{attribute addProperty BoxType "ELX3204-0000-0016"}
{attribute addProperty Id "RTD_Inputs_ChannelAT %I*ARRAY[0..3] OF RTD_Inputs_Channel_F16A160D128160WcStateAT %I*WcState_F855686C1620InfoDataAT %I*InfoData_BC63D37F80100"}
{attribute addProperty CRC "1009405569"}
{attribute addProperty SizeInBites "224"}
{attribute addProperty SizeInBytes "28"}
TYPE ELX3204_5DC9EB4C :
STRUCT
	{attribute addProperty Name "RTD_Inputs_Channel"}
	RTD_Inputs_Channel : ARRAY[0..3] OF RTD_Inputs_Channel_F16A160D;
	{attribute addProperty Name "WcState"}
	WcState : WcState_F855686C;
	{attribute addProperty Name "InfoData"}
	InfoData : InfoData_BC63D37F;
END_STRUCT
END_TYPE

(* stored: Version 1.2.0.0, ProductVersion 3.1.4024.9
   DUT ELX3204_5DC9EB4C: Id {df44a3c6-6b10-417a-be63-fc76bc59dbda} *)
